Staubli VAL3: start.pgx

program start()
begin
  movej(JApproach1,tToolSuccion, mNomSpeed)
  waitEndMove()
  movej(jGetCinta, tToolSuccion, mNomSpeed)
  waitEndMove()
  close(tToolSuccion)
  waitEndMove()
  movej(pApprBins, tToolSuccion, mNomSpeed)
  waitEndMove()
  open(tToolSuccion)
  waitEndMove()
end
